FUNCTION_BLOCK SCALE (* Scaling of an INT input to a UINT range of 0-100% *)
  (* Standard: 61499-1; Function: I/O *)
  (* Version 0.0, 2006-04-13, JHC, Holobloc Inc *)
  (* Compiler header: package fb.rt.process; *)
  (* Compiler Java Sun JDK 1.5.0 *)
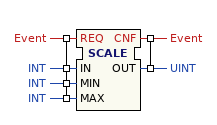
  EVENT_INPUT
    REQ WITH IN, MIN, MAX; (* Normal Execution Request *)
  END_EVENT
  EVENT_OUTPUT
    CNF WITH OUT; (* Execution Confirmation *)
  END_EVENT
  VAR_INPUT
    IN : INT; (* Process (typically A/D) input *)
    MIN : INT; (* IN value corresponding to OUT=0 *)
    MAX : INT; (* IN value corrsponding to OUT=100% *)
  END_VAR
  VAR_OUTPUT
    OUT : UINT; (* Scaled Output, limited to {0..100}% *)
  END_VAR
END_FUNCTION_BLOCK
